FUNCTION_BLOCK AXIS_REF_Ext EXTENDS AXIS_REF
VAR_INPUT
	EMG					:BOOL;
	Enable_Positive		:BOOL;
	Enable_Negative		:BOOL;
	AxisName			:STRING(50);
END_VAR
VAR_OUTPUT
	strAxisStates		:STRING(50);
	DI					AT %I* :UDINT;
	DeviceErrorcode			AT %I* :WORD;
END_VAR
VAR
	stEcSlaveAmsNetAdr 	AT %I* 			:ST_AmsAddr;
	_IndexCounter						:UDINT;
	MC_Power							:MC_Power;
	MC_Jog								:MC_Jog;
	_bSwich								:BOOL;
	_bJogFFlag,_bJogBFlag,_bStopFlag,_bResetFlag,_bMoveVelocityFlag,_bSetPosition			:BOOL;			//內部旗標 
	MC_Stop								:MC_Stop;
	MC_Reset							:MC_Reset;		
	MC_ReadParameter					:MC_ReadParameter;
	MC_ReadDriveAddress					:MC_ReadDriveAddress;
	MC_MoveVelocity						:MC_MoveVelocity;
	MC_SetPosition						:MC_SetPosition;
	MaxVelo								:LREAL;
	TempVelo							:LREAL;
	nJogStep,nStopStep,nResetStep,nMoveVelocityStep,nSetPositionStep		:INT;
	
	
	
END_VAR

SUPER^.ReadStatus();
SUPER^();
//flagtoString
AxisStatesToString();
/////////////////////////////////Power ON///////////////////////////////////
IF NOT EMG THEN
	_bSwich:=FALSE;
END_IF
MC_Power(
	Axis:= SUPER^, 
	Enable:= _bSwich, 
	Enable_Positive:= Enable_Positive, 
	Enable_Negative:= Enable_Negative, 
	Override:= , 
	BufferMode:= , 
	Options:= , 
	Status=> , 
	Busy=> , 
	Error=> , 
	ErrorID=> );
	
MC_ReadDriveAddress(
	Axis:= SUPER^, 
	Execute:= MC_Power.Status, 
	Done=> , 
	Busy=> , 
	Error=> , 
	ErrorID=> , 
	DriveAddress=> );	
	

///////////////////////////////////////////////////////////////
NStep();

ACTION AxisStatesToString:
CASE SUPER^.Status.MotionState OF
    MC_AXISSTATE_UNDEFINED:
		strAxisStates:='Undefined';
    MC_AXISSTATE_DISABLED:
		strAxisStates:='Disable';
    MC_AXISSTATE_STANDSTILL:
		strAxisStates:='Standstill';
    MC_AXISSTATE_ERRORSTOP:
		strAxisStates:='ErrorStop';
    MC_AXISSTATE_STOPPING:
		strAxisStates:='Stopping';
    MC_AXISSTATE_HOMING:
		strAxisStates:='Homing';
    MC_AXISSTATE_DISCRETEMOTION:
		strAxisStates:='Discretemotion';
    MC_AXISSTATE_CONTINOUSMOTION:
		strAxisStates:='Continousmotion';
    MC_AXISSTATE_SYNCHRONIZEDMOTION	:
		strAxisStates:='Synchronizedmotion';	
END_CASE
END_ACTION

PROPERTY CommandError : BOOL
GET
VAR
END_VAR
VAR_OUTPUT
	ErrorID	:	UDINT;
END_VAR
CommandError:= 	MC_Stop.Error OR MC_Reset.Error OR MC_Jog.Error OR MC_Power.Error OR MC_SetPosition.Error OR MC_MoveVelocity.Error;

ErrorID:=	MC_Stop.ErrorID OR MC_Reset.ErrorID OR MC_Jog.ErrorID OR MC_Power.ErrorID OR MC_SetPosition.ErrorID OR MC_MoveVelocity.ErrorID;
END_GET
END_PROPERTY

PROPERTY Error : BOOL
GET
Error:= SUPER^.Status.Error	OR  SUPER^.Status.DriveDeviceError;
END_GET
END_PROPERTY

METHOD JogBackwards : BOOL
VAR_INPUT
	Velocity: LREAL;
END_VAR
_bJogBFlag	:= TRUE;

IF NOT MC_Jog.JogForward THEN
	IF 	Velocity > MaxVelo THEN
		MC_Jog.Velocity	:= MaxVelo ; 
		ELSE
		MC_Jog.Velocity	:=	Velocity;
	END_IF
END_IF
JogBackwards:= SUPER^.Status.ConstantVelocity;
END_METHOD

METHOD JogForward : BOOL
VAR_INPUT
	Velocity	:LREAL;
END_VAR
_bJogFFlag	:= TRUE;

IF NOT MC_Jog.JogBackwards THEN
	IF 	Velocity > MaxVelo THEN
		MC_Jog.Velocity	:= MaxVelo ; 
		ELSE
		MC_Jog.Velocity	:=	Velocity;
	END_IF
END_IF
JogForward:= SUPER^.Status.ConstantVelocity;
END_METHOD

METHOD MoveVelocity : BOOL
VAR_INPUT
	Velocity			:LREAL;
	Direction 			:TC2_MC2.MC_Direction	 ;
(*MC_Positive_Direction := 1,MC_Shortest_Way ,MC_Negative_Direction,MC_Current_Direction,MC_Undefined_Direction := 128*)	
END_VAR
_bMoveVelocityFlag := TRUE;
TempVelo	:= Velocity ;
MC_MoveVelocity.Direction	:=  Direction;


MoveVelocity:= MC_MoveVelocity.InVelocity;
END_METHOD

ACTION NStep:
//////////////////////////////JOG//////////////////////////////////////	
MC_ReadParameter(
	Axis:= SUPER^, 
	Enable:=TRUE , 
	ParameterNumber:= MaxVelocitySystem, 
	ReadMode:=READMODE_CYCLIC , 
	Valid=> , 
	Busy=> , 
	Error=> , 
	ErrorID=> , 
	Value=> MaxVelo);
////////////////JOG+++//////////////////
MC_Jog(
	Axis:= SUPER^, 
	JogForward:= , 
	JogBackwards:= , 
	Mode:= MC_JOGMODE_CONTINOUS, 
	Position:= , 
	Velocity:= , 
	Acceleration:= , 
	Deceleration:= , 
	Jerk:= , 
	Done=> , 
	Busy=> , 
	Active=> , 
	CommandAborted=> , 
	Error=> , 
	ErrorID=> );
	
IF SUPER^.Status.Error THEN
	nJogStep:=0;
	_bJogFFlag:=FALSE;
	_bJogBFlag:=FALSE;
END_IF	
	
CASE nJogStep OF
	0:
		IF _bJogFFlag THEN
			IF SUPER^.Status.StandStill THEN
				nJogStep:= 10;
			END_IF;
		END_IF
		IF _bJogBFlag THEN
			IF SUPER^.Status.StandStill THEN
				nJogStep:= 15;
			END_IF;
		END_IF		
		
	10:
		MC_Jog.JogForward:=TRUE;
		IF NOT _bJogFFlag THEN
			MC_Jog.JogForward:=FALSE;
			nJogStep:= 0;
		END_IF	
		IF  SUPER^.Status.Stopping THEN
			MC_Jog.JogForward:=FALSE;
			nJogStep:= 20;		
		END_IF
		
	15:
		MC_Jog.JogBackwards:=TRUE;
		IF NOT _bJogBFlag THEN
			MC_Jog.JogBackwards:=FALSE;
			nJogStep:= 0;
		END_IF				
		IF  SUPER^.Status.Stopping THEN
			MC_Jog.JogBackwards:=FALSE;
			nJogStep:=20;		
		END_IF	
	20:
		IF NOT _bJogBFlag AND NOT _bJogFFlag THEN
			nJogStep:= 0;
		END_IF;
	
	50:
END_CASE	

	
_bJogFFlag:=FALSE;
_bJogBFlag:=FALSE;
//********************************************************
//STOP

MC_Stop(
	Axis:=SUPER^ , 
	Execute:= , 
	Deceleration:= , 
	Jerk:= , 
	Options:= , 
	Done=> , 
	Busy=> , 
	Active=> , 
	CommandAborted=> , 
	Error=> , 
	ErrorID=> );
CASE nStopStep OF
	0:	
		MC_Stop.Execute:= FALSE;
		IF _bStopFlag THEN
			MC_Stop.Execute:= TRUE;
			nStopStep	:= 10;	
		END_IF
	10:
		IF MC_Stop.Done THEN
			MC_Stop.Execute:= FALSE;
			nStopStep	:= 15;		
		END_IF;		
		IF MC_Stop.Error THEN
			MC_Stop.Execute:= FALSE;
			nStopStep	:= 20;		
		END_IF;	

		
	15:		
		IF NOT _bStopFlag THEN
			MC_Stop.Execute:= FALSE;
			nStopStep	:= 0;	
		END_IF	
	20:
		IF NOT _bStopFlag THEN
			MC_Stop.Execute:= FALSE;
			nStopStep	:= 0;	
		END_IF		
END_CASE;

_bStopFlag:=FALSE;
////////////////////////////////////////////////////
MC_Reset(Axis:=SUPER^);


CASE nResetStep OF
	0:	
		MC_Reset.Execute:= FALSE;
		IF _bResetFlag THEN
			MC_Reset.Execute:= TRUE;
			nResetStep	:= 10;	
		END_IF
	10:
		IF MC_Reset.Done THEN
			MC_Reset.Execute:= FALSE;
			nResetStep	:= 15;		
		END_IF;		
		IF MC_Reset.Error THEN
			MC_Reset.Execute:= FALSE;
			nResetStep	:= 20;		
		END_IF;	

		
	15:		
		IF NOT _bResetFlag THEN
			nResetStep	:= 0;	
		END_IF	
	20:
		IF NOT _bResetFlag THEN
			nResetStep	:= 0;	
		END_IF	
	
END_CASE;


	
_bResetFlag	:=FALSE;
////////////////////////////////////////////////////////////////////	
MC_MoveVelocity(Axis:= SUPER^);
IF SUPER^.Status.Error  THEN
	nMoveVelocityStep	:= 0;
END_IF

CASE nMoveVelocityStep OF
	0:	
		MC_MoveVelocity.Execute:= FALSE;
		IF _bMoveVelocityFlag AND SUPER^.Status.StandStill AND NOT SUPER^.Status.Error  THEN
			MC_MoveVelocity.Velocity	:= TempVelo;
			MC_MoveVelocity.Execute:= TRUE;
			nMoveVelocityStep	:= 5;
		END_IF
	
	5:
		IF MC_MoveVelocity.Velocity	<> TempVelo THEN
			MC_MoveVelocity.Execute:= FALSE;
			nMoveVelocityStep	:= 6;
		END_IF
		IF NOT _bMoveVelocityFlag THEN
			nMoveVelocityStep	:= 20;
		END_IF
	6:
		IF NOT MC_MoveVelocity.Active THEN
			MC_MoveVelocity.Velocity	:= TempVelo;
			MC_MoveVelocity.Execute		:= TRUE;
			nMoveVelocityStep			:= 5;
		END_IF;		

	20:
		IF Stop() THEN
			nMoveVelocityStep	:= 0;
		END_IF		
	
END_CASE;	
_bMoveVelocityFlag := FALSE;

//////////////////////////////////////////////////////////////
MC_SetPosition(Axis:= SUPER^);
CASE nSetPositionStep OF
	0:
		MC_SetPosition.Execute:= FALSE;
		IF _bSetPosition THEN
			MC_SetPosition.Execute:= TRUE;
			nSetPositionStep:= 5;
		END_IF
	
	5:
		IF MC_SetPosition.Done THEN
			nSetPositionStep:= 10;
		END_IF
		IF MC_SetPosition.Error THEN
			nSetPositionStep:= 15;
		END_IF
	10:
		IF NOT _bSetPosition THEN
			MC_SetPosition.Execute:= FALSE;
			nSetPositionStep:= 0;
		END_IF
	15:
		IF NOT _bSetPosition THEN
			MC_SetPosition.Execute:= FALSE;
			nSetPositionStep:= 0;
		END_IF

END_CASE






_bSetPosition	:=FALSE;
END_ACTION

METHOD Reset : BOOL
VAR_INPUT
END_VAR
_bResetFlag	:=TRUE;
Reset := nResetStep = 15;
END_METHOD

METHOD ServoOFF : BOOL
VAR_INPUT
END_VAR
_bSwich	:= FALSE;
ServoOFF	:= SUPER^.Status.Disabled;
END_METHOD

METHOD ServoOn : BOOL
VAR_INPUT
END_VAR
IF EMG THEN
	_bSwich	:= TRUE;
	ELSE
	_bSwich	:= FALSE;
END_IF
ServoOn := MC_Power.Status;
END_METHOD

METHOD SetPosition : BOOL
VAR_INPUT
	Position:LREAL;
END_VAR
_bSetPosition	:=TRUE;
MC_SetPosition.Position:= Position;

SetPosition	:= MC_SetPosition.Done;
END_METHOD

METHOD Stop : BOOL
VAR_INPUT
END_VAR
_bStopFlag	:= TRUE;
Stop:=  nStopStep=15 ;
END_METHOD

END_FUNCTION_BLOCK

(* stored: Version 1.1.0.1, ProductVersion 3.1.4024.16
   POU AXIS_REF_Ext: Id {32eaf42d-4ad2-4a2f-948a-ee8f04bd528b}, SpecialFunc None
   Action AxisStatesToString: Id {75afc977-fac9-4914-ba48-9b3fbee98525}
   Property CommandError: Id {fff79de0-3f0d-493f-b350-dc0661c29af5}
   Get Get: Id {40482807-0ec2-4f85-a612-a6c4bc555d37}
   Property Error: Id {5a1a4e2d-9c31-4c08-a963-a89633d6cf02}
   Get Get: Id {6959e72b-1603-4476-8751-49b38779cc1e}
   Method JogBackwards: Id {4371965c-c41a-4c36-9506-740d0e6bc726}
   Method JogForward: Id {fe1c87ad-4f62-40d5-ae18-3038a701af3c}
   Method MoveVelocity: Id {74e4f9de-6438-447f-8fd0-707f0926bd22}
   Action NStep: Id {8c16e0d9-aa4f-4123-af8f-dce3d8db2ceb}
   Method Reset: Id {5d069d86-3ec8-4e54-8284-e7151190a704}
   Method ServoOFF: Id {a56c4bf4-f3f6-4623-8441-2f08556512bf}
   Method ServoOn: Id {bcad41ad-1d48-4fe7-a7cd-07bdf8658b01}
   Method SetPosition: Id {ae728b18-df04-4a9e-bade-cabf4ce9bbc3}
   Method Stop: Id {c508e04b-7649-4e5d-a07a-20ec63583a85} *)
